// TIA Portal project "Progetto_Packaging_Process" (V16)

(* hardware
DEVICE "S7-1200 station_1"  S7-1200 Station
   slot 0: "Telaio di montaggio_0"  S7-1200 Rack  Rack  V1.0
   slot 1: "PLC_1"  CPU 1212C AC/DC/Rly  6ES7 212-1BE40-0XB0  V4.4
*)

// ===== PLC "PLC_1"  CPU 1212C AC/DC/Rly =====

VAR_GLOBAL   // PLC tag table "Tabella delle variabili standard"
   "System_Byte" AT %MB1 : Byte;
   "FirstScan" AT %M1.0 : Bool;
   "DiagStatusUpdate" AT %M1.1 : Bool;
   "AlwaysTRUE" AT %M1.2 : Bool;
   "AlwaysFALSE" AT %M1.3 : Bool;
   "System_Byte(1)" AT %MB1 : Byte;
   "System_Byte(2)" AT %MB1 : Byte;
   "Clock_Byte" AT %MB0 : Byte;
   "Clock_10Hz" AT %M0.0 : Bool;
   "Clock_5Hz" AT %M0.1 : Bool;
   "Clock_2.5Hz" AT %M0.2 : Bool;
   "Clock_2Hz" AT %M0.3 : Bool;
   "Clock_1.25Hz" AT %M0.4 : Bool;
   "Clock_1Hz" AT %M0.5 : Bool;
   "Clock_0.625Hz" AT %M0.6 : Bool;
   "Clock_0.5Hz" AT %M0.7 : Bool;
   "Start" AT %I0.0 : Bool;
   "Stop" AT %I0.1 : Bool;
   "Emergency Stop" AT %I0.2 : Bool;
   "Pacco vuoto" AT %I0.3 : Bool;
   "Plastica 1" AT %I0.4 : Bool;
   "Oggetto" AT %I0.5 : Bool;
   "Plastica 2" AT %I0.6 : Bool;
   "Chiusura Alette" AT %I0.7 : Bool;
   "Scotch" AT %I1.0 : Bool;
   "Postazione di peso" AT %I1.1 : Bool;
   "Sensore di peso" AT %I1.2 : Bool;
   "Pacco Smistato" AT %I1.3 : Bool;
   "Conveyor Pacchi vuoti" AT %Q0.0 : Bool;
   "Conveyor Principale" AT %Q0.1 : Bool;
   "Conveyor Oggetti" AT %Q0.2 : Bool;
   "Conveyor Smistamento" AT %Q0.3 : Bool;
   "Braccio Plastica" AT %Q0.4 : Bool;
   "Braccio Scotch" AT %Q0.5 : Bool;
   "Pedana di peso" AT %Q0.6 : Bool;
   "Guida Sx" AT %Q0.7 : Bool;
   "Guida Dx" AT %Q1.0 : Bool;
   "Luce sistema spento" AT %Q1.1 : Bool;
   "Luce pacco in movimento" AT %Q1.2 : Bool;
   "Luce pacco in lavorazione" AT %Q1.3 : Bool;
   "Stato 0" AT %M2.0 : Bool;
   "Stato 1" AT %M2.1 : Bool;
   "Stato 2" AT %M2.2 : Bool;
   "Stato 3" AT %M2.3 : Bool;
   "Stato 4" AT %M2.4 : Bool;
   "Stato 5" AT %M2.5 : Bool;
   "Stato 6" AT %M2.6 : Bool;
   "Stato 7" AT %M2.7 : Bool;
   "Stato 8" AT %M3.0 : Bool;
   "Stato 9" AT %M3.1 : Bool;
   "Stato 10" AT %M3.2 : Bool;
   "Stato 11" AT %M3.3 : Bool;
   "Stato 12" AT %M3.4 : Bool;
   "Tag_1" AT %Q1.4 : Bool;
END_VAR

// folder: System blocks/Program resources

DATA_BLOCK "T1"   // DB1
{ S7_Optimized_Access := 'TRUE' }
AUTHOR : Simatic
FAMILY : IEC
NAME : IEC_TMR
VERSION : 1.0
// stored: InstanceOfName IEC_TIMER
"IEC_TIMER"
BEGIN
END_DATA_BLOCK

DATA_BLOCK "T2"   // DB2
{ S7_Optimized_Access := 'TRUE' }
AUTHOR : Simatic
FAMILY : IEC
NAME : IEC_TMR
VERSION : 1.0
// stored: InstanceOfName IEC_TIMER
"IEC_TIMER"
BEGIN
END_DATA_BLOCK

DATA_BLOCK "T3"   // DB3
{ S7_Optimized_Access := 'TRUE' }
AUTHOR : Simatic
FAMILY : IEC
NAME : IEC_TMR
VERSION : 1.0
// stored: InstanceOfName IEC_TIMER
"IEC_TIMER"
BEGIN
END_DATA_BLOCK

DATA_BLOCK "CNT2"   // DB4
{ S7_Optimized_Access := 'TRUE' }
AUTHOR : Simatic
FAMILY : IEC
NAME : CNTR
VERSION : 1.0
// stored: InstanceOfName IEC_COUNTER
"IEC_COUNTER"
BEGIN
END_DATA_BLOCK

DATA_BLOCK "CNT1"   // DB5
{ S7_Optimized_Access := 'TRUE' }
AUTHOR : Simatic
FAMILY : IEC
NAME : CNTR
VERSION : 1.0
// stored: InstanceOfName IEC_COUNTER
"IEC_COUNTER"
BEGIN
END_DATA_BLOCK

// folder: (top level)

ORGANIZATION_BLOCK "Main"   // OB1, LAD, ProgramCycle
TITLE = "Main Program Sweep (Cycle)" / Automation product packaging process
{ S7_Optimized_Access := 'TRUE' }
VERSION : 0.1
   VAR_INPUT
      Initial_Call : Bool;   // Initial call of this OB
      Remanence : Bool;   // =True, if remanent data are available
   END_VAR
   VAR_TEMP   // added for the SCL form of the ladder/FBD networks
      _w1 : Bool;
   END_VAR
BEGIN

REGION Network 1: Inizializzazione
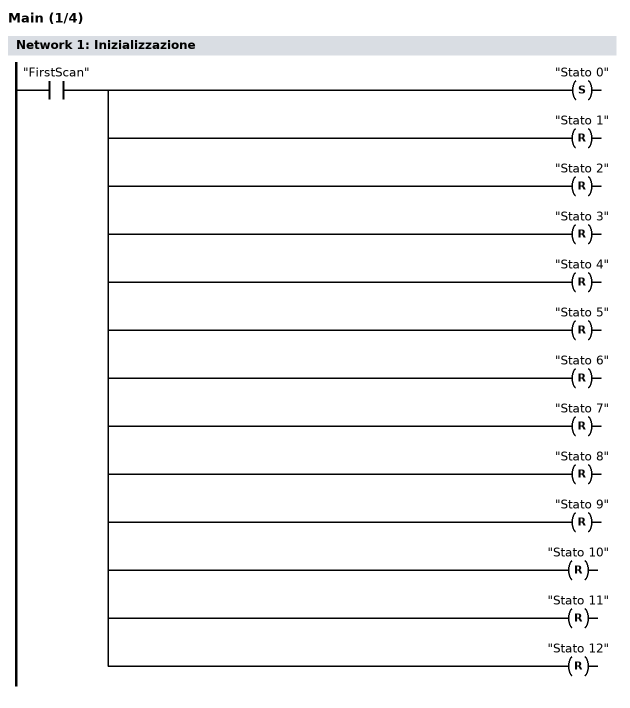
   RUNG wire#powerrail
      Contact( "FirstScan" )
      wire#w1
      S_Coil( "Stato 0" )
   END_RUNG
   RUNG wire#w1
      R_Coil( "Stato 1" )
   END_RUNG
   RUNG wire#w1
      R_Coil( "Stato 2" )
   END_RUNG
   RUNG wire#w1
      R_Coil( "Stato 3" )
   END_RUNG
   RUNG wire#w1
      R_Coil( "Stato 4" )
   END_RUNG
   RUNG wire#w1
      R_Coil( "Stato 5" )
   END_RUNG
   RUNG wire#w1
      R_Coil( "Stato 6" )
   END_RUNG
   RUNG wire#w1
      R_Coil( "Stato 7" )
   END_RUNG
   RUNG wire#w1
      R_Coil( "Stato 8" )
   END_RUNG
   RUNG wire#w1
      R_Coil( "Stato 9" )
   END_RUNG
   RUNG wire#w1
      R_Coil( "Stato 10" )
   END_RUNG
   RUNG wire#w1
      R_Coil( "Stato 11" )
   END_RUNG
   RUNG wire#w1
      R_Coil( "Stato 12" )
   END_RUNG
   // the same network as SCL:
   IF "FirstScan" THEN
       "Stato 0" := TRUE;
       "Stato 1" := FALSE;
       "Stato 2" := FALSE;
       "Stato 3" := FALSE;
       "Stato 4" := FALSE;
       "Stato 5" := FALSE;
       "Stato 6" := FALSE;
       "Stato 7" := FALSE;
       "Stato 8" := FALSE;
       "Stato 9" := FALSE;
       "Stato 10" := FALSE;
       "Stato 11" := FALSE;
       "Stato 12" := FALSE;
   END_IF;
END_REGION

REGION Network 2: Transizioni
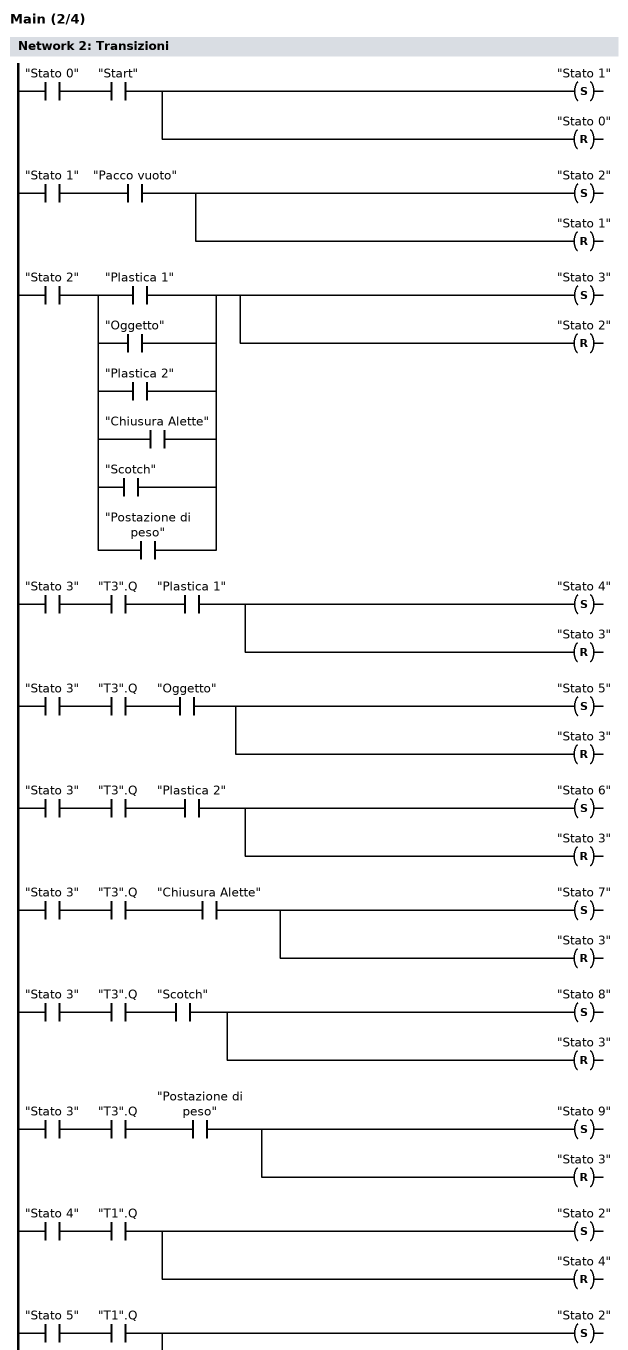
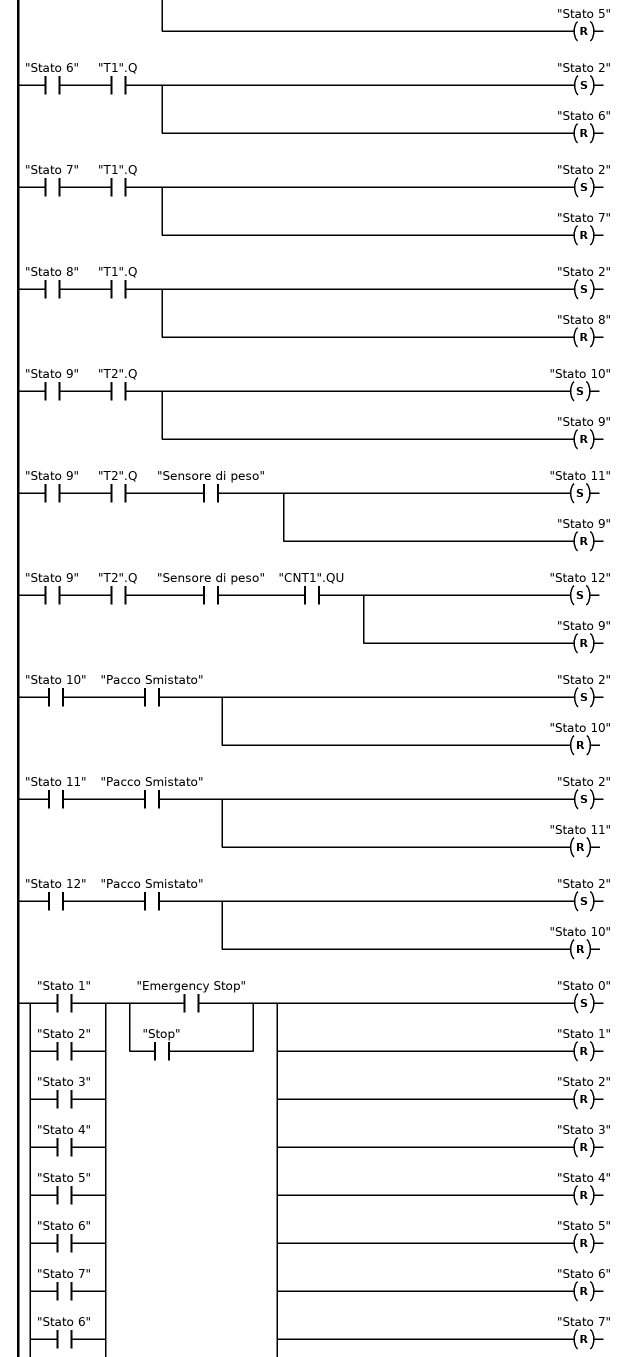
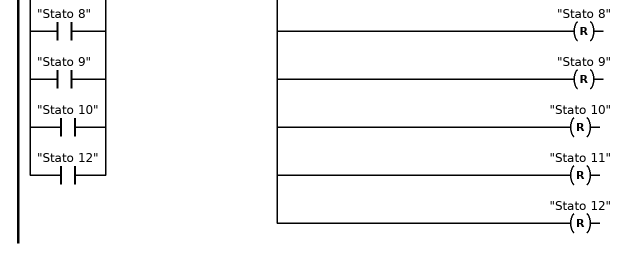
   RUNG wire#powerrail
      Contact( "Stato 0" )
      Contact( "Start" )
      wire#w1
      S_Coil( "Stato 1" )
   END_RUNG
   RUNG wire#w1
      R_Coil( "Stato 0" )
   END_RUNG
   RUNG wire#powerrail
      Contact( "Stato 1" )
      Contact( "Pacco vuoto" )
      wire#w2
      S_Coil( "Stato 2" )
   END_RUNG
   RUNG wire#w2
      R_Coil( "Stato 1" )
   END_RUNG
   RUNG wire#powerrail
      Contact( "Stato 2" )
      wire#w3
      Contact( "Plastica 1" )
      wire#w4
      S_Coil( "Stato 3" )
   END_RUNG
   RUNG wire#w3
      Contact( "Oggetto" )
   END_RUNG wire#w4
   RUNG wire#w3
      Contact( "Plastica 2" )
   END_RUNG wire#w4
   RUNG wire#w3
      Contact( "Chiusura Alette" )
   END_RUNG wire#w4
   RUNG wire#w3
      Contact( "Scotch" )
   END_RUNG wire#w4
   RUNG wire#w3
      Contact( "Postazione di peso" )
   END_RUNG wire#w4
   RUNG wire#w4
      R_Coil( "Stato 2" )
   END_RUNG
   RUNG wire#powerrail
      Contact( "Stato 3" )
      Contact( "T3".Q )
      Contact( "Plastica 1" )
      wire#w5
      S_Coil( "Stato 4" )
   END_RUNG
   RUNG wire#w5
      R_Coil( "Stato 3" )
   END_RUNG
   RUNG wire#powerrail
      Contact( "Stato 3" )
      Contact( "T3".Q )
      Contact( "Oggetto" )
      wire#w6
      S_Coil( "Stato 5" )
   END_RUNG
   RUNG wire#w6
      R_Coil( "Stato 3" )
   END_RUNG
   RUNG wire#powerrail
      Contact( "Stato 3" )
      Contact( "T3".Q )
      Contact( "Plastica 2" )
      wire#w7
      S_Coil( "Stato 6" )
   END_RUNG
   RUNG wire#w7
      R_Coil( "Stato 3" )
   END_RUNG
   RUNG wire#powerrail
      Contact( "Stato 3" )
      Contact( "T3".Q )
      Contact( "Chiusura Alette" )
      wire#w8
      S_Coil( "Stato 7" )
   END_RUNG
   RUNG wire#w8
      R_Coil( "Stato 3" )
   END_RUNG
   RUNG wire#powerrail
      Contact( "Stato 3" )
      Contact( "T3".Q )
      Contact( "Scotch" )
      wire#w9
      S_Coil( "Stato 8" )
   END_RUNG
   RUNG wire#w9
      R_Coil( "Stato 3" )
   END_RUNG
   RUNG wire#powerrail
      Contact( "Stato 3" )
      Contact( "T3".Q )
      Contact( "Postazione di peso" )
      wire#w10
      S_Coil( "Stato 9" )
   END_RUNG
   RUNG wire#w10
      R_Coil( "Stato 3" )
   END_RUNG
   RUNG wire#powerrail
      Contact( "Stato 4" )
      Contact( "T1".Q )
      wire#w11
      S_Coil( "Stato 2" )
   END_RUNG
   RUNG wire#w11
      R_Coil( "Stato 4" )
   END_RUNG
   RUNG wire#powerrail
      Contact( "Stato 5" )
      Contact( "T1".Q )
      wire#w12
      S_Coil( "Stato 2" )
   END_RUNG
   RUNG wire#w12
      R_Coil( "Stato 5" )
   END_RUNG
   RUNG wire#powerrail
      Contact( "Stato 6" )
      Contact( "T1".Q )
      wire#w13
      S_Coil( "Stato 2" )
   END_RUNG
   RUNG wire#w13
      R_Coil( "Stato 6" )
   END_RUNG
   RUNG wire#powerrail
      Contact( "Stato 7" )
      Contact( "T1".Q )
      wire#w14
      S_Coil( "Stato 2" )
   END_RUNG
   RUNG wire#w14
      R_Coil( "Stato 7" )
   END_RUNG
   RUNG wire#powerrail
      Contact( "Stato 8" )
      Contact( "T1".Q )
      wire#w15
      S_Coil( "Stato 2" )
   END_RUNG
   RUNG wire#w15
      R_Coil( "Stato 8" )
   END_RUNG
   RUNG wire#powerrail
      Contact( "Stato 9" )
      Contact( "T2".Q )
      wire#w16
      S_Coil( "Stato 10" )
   END_RUNG
   RUNG wire#w16
      R_Coil( "Stato 9" )
   END_RUNG
   RUNG wire#powerrail
      Contact( "Stato 9" )
      Contact( "T2".Q )
      Contact( "Sensore di peso" )
      wire#w17
      S_Coil( "Stato 11" )
   END_RUNG
   RUNG wire#w17
      R_Coil( "Stato 9" )
   END_RUNG
   RUNG wire#powerrail
      Contact( "Stato 9" )
      Contact( "T2".Q )
      Contact( "Sensore di peso" )
      Contact( "CNT1".QU )
      wire#w18
      S_Coil( "Stato 12" )
   END_RUNG
   RUNG wire#w18
      R_Coil( "Stato 9" )
   END_RUNG
   RUNG wire#powerrail
      Contact( "Stato 10" )
      Contact( "Pacco Smistato" )
      wire#w19
      S_Coil( "Stato 2" )
   END_RUNG
   RUNG wire#w19
      R_Coil( "Stato 10" )
   END_RUNG
   RUNG wire#powerrail
      Contact( "Stato 11" )
      Contact( "Pacco Smistato" )
      wire#w20
      S_Coil( "Stato 2" )
   END_RUNG
   RUNG wire#w20
      R_Coil( "Stato 11" )
   END_RUNG
   RUNG wire#powerrail
      Contact( "Stato 12" )
      Contact( "Pacco Smistato" )
      wire#w21
      S_Coil( "Stato 2" )
   END_RUNG
   RUNG wire#w21
      R_Coil( "Stato 10" )
   END_RUNG
   RUNG wire#powerrail
      Contact( "Stato 1" )
      wire#w22
      Contact( "Emergency Stop" )
      wire#w23
      S_Coil( "Stato 0" )
   END_RUNG
   RUNG wire#powerrail
      Contact( "Stato 2" )
   END_RUNG wire#w22
   RUNG wire#powerrail
      Contact( "Stato 3" )
   END_RUNG wire#w22
   RUNG wire#powerrail
      Contact( "Stato 4" )
   END_RUNG wire#w22
   RUNG wire#powerrail
      Contact( "Stato 5" )
   END_RUNG wire#w22
   RUNG wire#powerrail
      Contact( "Stato 6" )
   END_RUNG wire#w22
   RUNG wire#powerrail
      Contact( "Stato 7" )
   END_RUNG wire#w22
   RUNG wire#powerrail
      Contact( "Stato 6" )
   END_RUNG wire#w22
   RUNG wire#powerrail
      Contact( "Stato 8" )
   END_RUNG wire#w22
   RUNG wire#powerrail
      Contact( "Stato 9" )
   END_RUNG wire#w22
   RUNG wire#powerrail
      Contact( "Stato 10" )
   END_RUNG wire#w22
   RUNG wire#powerrail
      Contact( "Stato 12" )
   END_RUNG wire#w22
   RUNG wire#w22
      Contact( "Stop" )
   END_RUNG wire#w23
   RUNG wire#w23
      R_Coil( "Stato 1" )
   END_RUNG
   RUNG wire#w23
      R_Coil( "Stato 2" )
   END_RUNG
   RUNG wire#w23
      R_Coil( "Stato 3" )
   END_RUNG
   RUNG wire#w23
      R_Coil( "Stato 4" )
   END_RUNG
   RUNG wire#w23
      R_Coil( "Stato 5" )
   END_RUNG
   RUNG wire#w23
      R_Coil( "Stato 6" )
   END_RUNG
   RUNG wire#w23
      R_Coil( "Stato 7" )
   END_RUNG
   RUNG wire#w23
      R_Coil( "Stato 8" )
   END_RUNG
   RUNG wire#w23
      R_Coil( "Stato 9" )
   END_RUNG
   RUNG wire#w23
      R_Coil( "Stato 10" )
   END_RUNG
   RUNG wire#w23
      R_Coil( "Stato 11" )
   END_RUNG
   RUNG wire#w23
      R_Coil( "Stato 12" )
   END_RUNG
   // the same network as SCL:
   IF "Stato 0" AND "Start" THEN
       "Stato 1" := TRUE;
       "Stato 0" := FALSE;
   END_IF;
   IF "Stato 1" AND "Pacco vuoto" THEN
       "Stato 2" := TRUE;
       "Stato 1" := FALSE;
   END_IF;
   IF "Stato 2" AND ("Plastica 1" OR "Oggetto" OR "Plastica 2" OR "Chiusura Alette" OR "Scotch" OR "Postazione di peso") THEN
       "Stato 3" := TRUE;
       "Stato 2" := FALSE;
   END_IF;
   IF "Stato 3" AND "T3".Q AND "Plastica 1" THEN
       "Stato 4" := TRUE;
       "Stato 3" := FALSE;
   END_IF;
   IF "Stato 3" AND "T3".Q AND "Oggetto" THEN
       "Stato 5" := TRUE;
       "Stato 3" := FALSE;
   END_IF;
   IF "Stato 3" AND "T3".Q AND "Plastica 2" THEN
       "Stato 6" := TRUE;
       "Stato 3" := FALSE;
   END_IF;
   IF "Stato 3" AND "T3".Q AND "Chiusura Alette" THEN
       "Stato 7" := TRUE;
       "Stato 3" := FALSE;
   END_IF;
   IF "Stato 3" AND "T3".Q AND "Scotch" THEN
       "Stato 8" := TRUE;
       "Stato 3" := FALSE;
   END_IF;
   IF "Stato 3" AND "T3".Q AND "Postazione di peso" THEN
       "Stato 9" := TRUE;
       "Stato 3" := FALSE;
   END_IF;
   IF "Stato 4" AND "T1".Q THEN
       "Stato 2" := TRUE;
       "Stato 4" := FALSE;
   END_IF;
   IF "Stato 5" AND "T1".Q THEN
       "Stato 2" := TRUE;
       "Stato 5" := FALSE;
   END_IF;
   IF "Stato 6" AND "T1".Q THEN
       "Stato 2" := TRUE;
       "Stato 6" := FALSE;
   END_IF;
   IF "Stato 7" AND "T1".Q THEN
       "Stato 2" := TRUE;
       "Stato 7" := FALSE;
   END_IF;
   IF "Stato 8" AND "T1".Q THEN
       "Stato 2" := TRUE;
       "Stato 8" := FALSE;
   END_IF;
   IF "Stato 9" AND "T2".Q THEN
       "Stato 10" := TRUE;
       "Stato 9" := FALSE;
   END_IF;
   IF "Stato 9" AND "T2".Q AND "Sensore di peso" THEN
       "Stato 11" := TRUE;
       "Stato 9" := FALSE;
   END_IF;
   IF "Stato 9" AND "T2".Q AND "Sensore di peso" AND "CNT1".QU THEN
       "Stato 12" := TRUE;
       "Stato 9" := FALSE;
   END_IF;
   IF "Stato 10" AND "Pacco Smistato" THEN
       "Stato 2" := TRUE;
       "Stato 10" := FALSE;
   END_IF;
   IF "Stato 11" AND "Pacco Smistato" THEN
       "Stato 2" := TRUE;
       "Stato 11" := FALSE;
   END_IF;
   IF "Stato 12" AND "Pacco Smistato" THEN
       "Stato 2" := TRUE;
       "Stato 10" := FALSE;
   END_IF;
   IF ("Stato 1" OR "Stato 2" OR "Stato 3" OR "Stato 4" OR "Stato 5" OR "Stato 6" OR "Stato 7" OR "Stato 6" OR "Stato 8" OR "Stato 9" OR "Stato 10" OR "Stato 12") AND ("Emergency Stop" OR "Stop") THEN
       "Stato 0" := TRUE;
   END_IF;
   #_w1 := ("Stato 1" OR "Stato 2" OR "Stato 3" OR "Stato 4" OR "Stato 5" OR "Stato 6" OR "Stato 7" OR "Stato 6" OR "Stato 8" OR "Stato 9" OR "Stato 10" OR "Stato 12") AND ("Emergency Stop" OR "Stop");
   IF #_w1 THEN
       "Stato 1" := FALSE;
       "Stato 2" := FALSE;
       "Stato 3" := FALSE;
       "Stato 4" := FALSE;
       "Stato 5" := FALSE;
       "Stato 6" := FALSE;
       "Stato 7" := FALSE;
       "Stato 8" := FALSE;
       "Stato 9" := FALSE;
       "Stato 10" := FALSE;
       "Stato 11" := FALSE;
       "Stato 12" := FALSE;
   END_IF;
END_REGION

REGION Network 3: Comandi
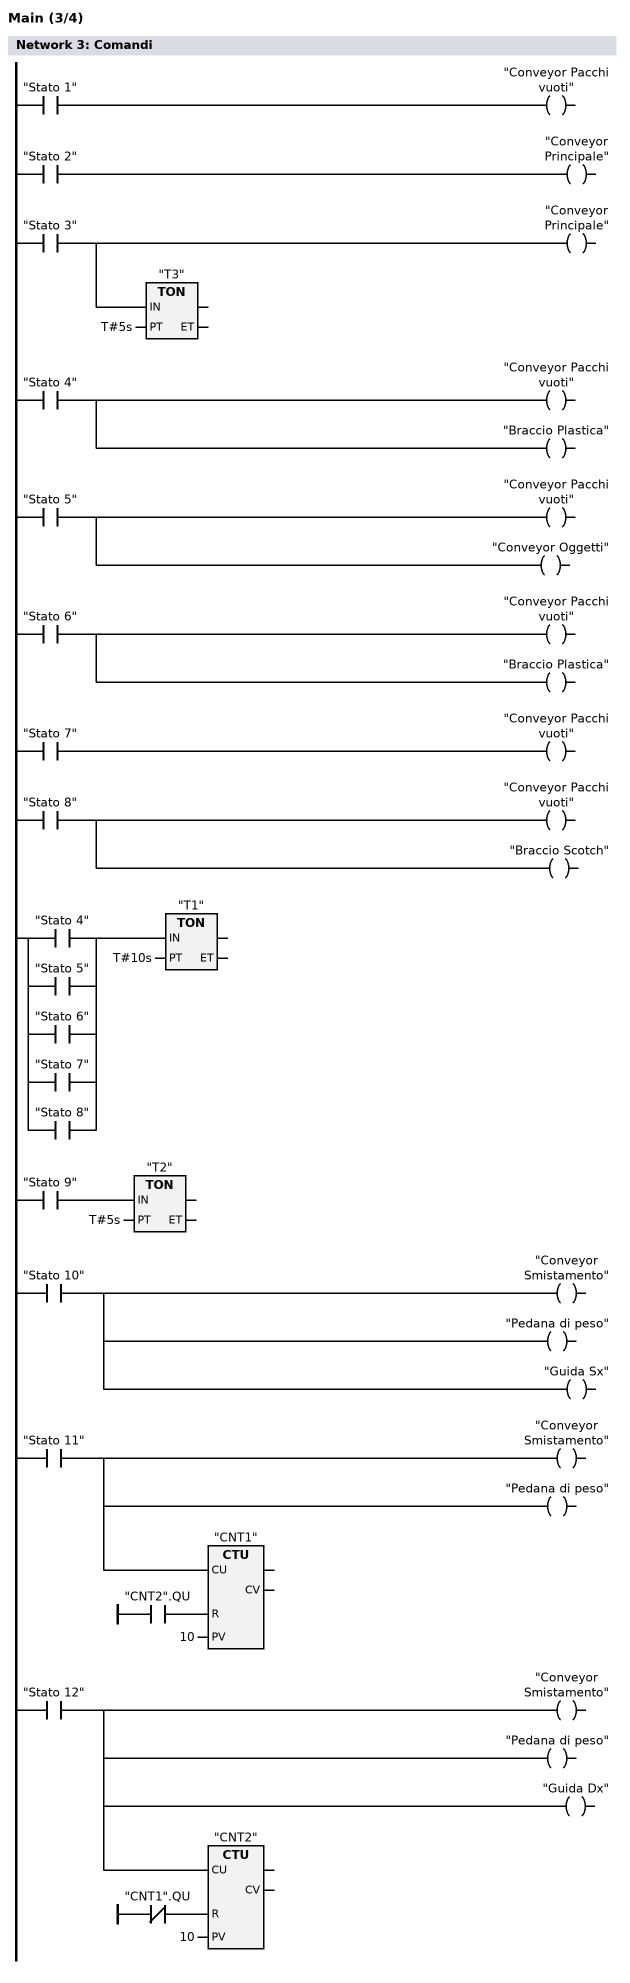
   "Conveyor Pacchi vuoti" := "Stato 1";
   "Conveyor Principale" := "Stato 2";
   "Conveyor Principale" := "Stato 3";
   "T3".TON(IN := "Stato 3", PT := T#5s);
   "Conveyor Pacchi vuoti" := "Stato 4";
   "Braccio Plastica" := "Stato 4";
   "Conveyor Pacchi vuoti" := "Stato 5";
   "Conveyor Oggetti" := "Stato 5";
   "Conveyor Pacchi vuoti" := "Stato 6";
   "Braccio Plastica" := "Stato 6";
   "Conveyor Pacchi vuoti" := "Stato 7";
   "Conveyor Pacchi vuoti" := "Stato 8";
   "Braccio Scotch" := "Stato 8";
   "T1".TON(IN := "Stato 4" OR "Stato 5" OR "Stato 6" OR "Stato 7" OR "Stato 8", PT := T#10s);
   "T2".TON(IN := "Stato 9", PT := T#5s);
   "Conveyor Smistamento" := "Stato 10";
   "Pedana di peso" := "Stato 10";
   "Guida Sx" := "Stato 10";
   "Conveyor Smistamento" := "Stato 11";
   "Pedana di peso" := "Stato 11";
   "CNT1".CTU(CU := "Stato 11", R := "CNT2".QU, PV := 10);
   "Conveyor Smistamento" := "Stato 12";
   "Pedana di peso" := "Stato 12";
   "Guida Dx" := "Stato 12";
   "CNT2".CTU(CU := "Stato 12", R := NOT "CNT1".QU, PV := 10);
END_REGION

REGION Network 4: Segnali Luminosi
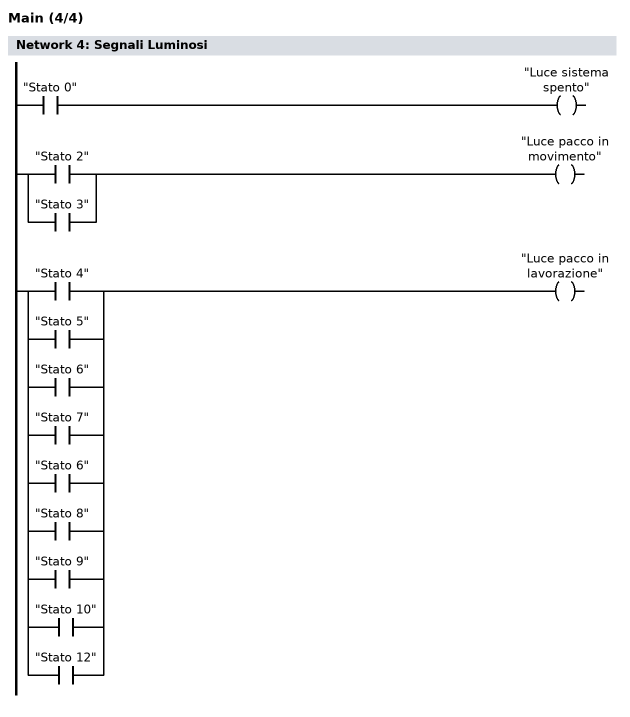
   RUNG wire#powerrail
      Contact( "Stato 0" )
      Coil( "Luce sistema spento" )
   END_RUNG
   RUNG wire#powerrail
      Contact( "Stato 2" )
      wire#w1
      Coil( "Luce pacco in movimento" )
   END_RUNG
   RUNG wire#powerrail
      Contact( "Stato 3" )
   END_RUNG wire#w1
   RUNG wire#powerrail
      Contact( "Stato 4" )
      wire#w2
      Coil( "Luce pacco in lavorazione" )
   END_RUNG
   RUNG wire#powerrail
      Contact( "Stato 5" )
   END_RUNG wire#w2
   RUNG wire#powerrail
      Contact( "Stato 6" )
   END_RUNG wire#w2
   RUNG wire#powerrail
      Contact( "Stato 7" )
   END_RUNG wire#w2
   RUNG wire#powerrail
      Contact( "Stato 6" )
   END_RUNG wire#w2
   RUNG wire#powerrail
      Contact( "Stato 8" )
   END_RUNG wire#w2
   RUNG wire#powerrail
      Contact( "Stato 9" )
   END_RUNG wire#w2
   RUNG wire#powerrail
      Contact( "Stato 10" )
   END_RUNG wire#w2
   RUNG wire#powerrail
      Contact( "Stato 12" )
   END_RUNG wire#w2
   // the same network as SCL:
   "Luce sistema spento" := "Stato 0";
   "Luce pacco in movimento" := "Stato 2" OR "Stato 3";
   "Luce pacco in lavorazione" := "Stato 4" OR "Stato 5" OR "Stato 6" OR "Stato 7" OR "Stato 6" OR "Stato 8" OR "Stato 9" OR "Stato 10" OR "Stato 12";
END_REGION
END_ORGANIZATION_BLOCK